FUNCTION_BLOCK FB_LEN (* IEC 61131-3,Table 29#1 *)
  (* Standard: IEC 61499 *)
  (* Version 0.1, 2006-09-15, JHC, Holobloc Inc, Moved to fb.rt.strings. *)
  (* Version 0.0, 2004-12-15, JHC, Rockwell Automation, Converted from SRC format. *)
  (* Compiler header: package fb.rt.strings; *)
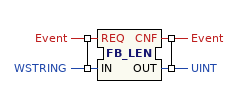
  EVENT_INPUT
    REQ WITH IN;
  END_EVENT
  EVENT_OUTPUT
    CNF WITH OUT;
  END_EVENT
  VAR_INPUT
    IN : WSTRING;
  END_VAR
  VAR_OUTPUT
    OUT : UINT;
  END_VAR
END_FUNCTION_BLOCK
